FUNCTION_BLOCK FB_SetResetFallTrigger
VAR_IN_OUT
	bVariable		: BOOL;
END_VAR
VAR_INPUT
	bSetResetTrigger	: BOOL;
END_VAR
VAR_OUTPUT
END_VAR
VAR
	trigger	: F_TRIG;
	reset	: RS;
END_VAR
VAR // added by the converter: edge detectors and wires of the graphical bodies
    _w1 : BOOL;
END_VAR

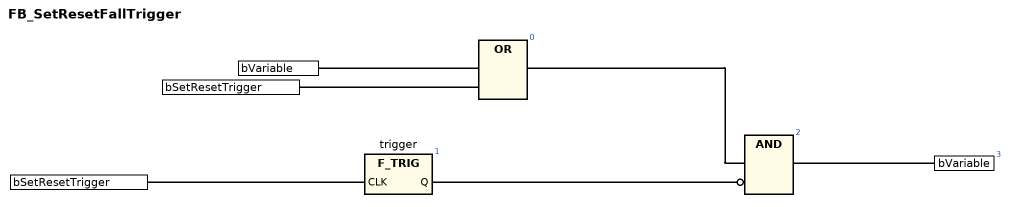
_w1 := bVariable OR bSetResetTrigger;
trigger(CLK := bSetResetTrigger); // F_TRIG
bVariable := _w1 AND NOT trigger.Q;

END_FUNCTION_BLOCK

(* stored: Version 1.1.0.1, ProductVersion 3.1.4024.9
   POU FB_SetResetFallTrigger: Id {24a786ad-5f6c-48cb-af83-9b9f7c6716b4}, SpecialFunc None *)
